PROGRAM PG_Regen
VAR
	Regenmacher: FB_Regenmacher;;
	Wetterbericht: FB_Wetterbericht;
END_VAR
VAR // added by the converter: edge detectors and wires of the graphical bodies
    _w1 : ANY;
END_VAR

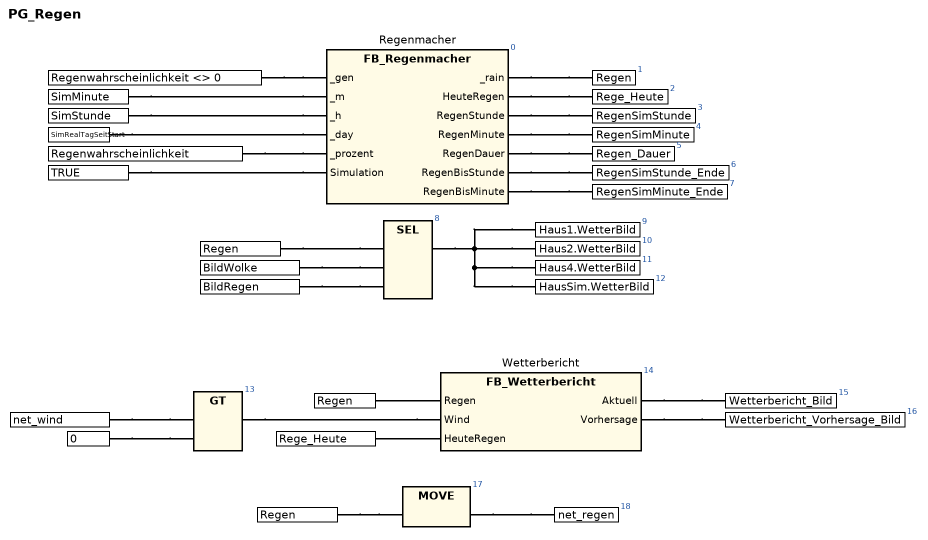
Regenmacher(
    _gen := Regenwahrscheinlichkeit <> 0,
    _m := SimMinute,
    _h := SimStunde,
    _day := SimRealTagSeitStart,
    _prozent := Regenwahrscheinlichkeit,
    Simulation := TRUE); // FB_Regenmacher
Regen := Regenmacher._rain;
Rege_Heute := Regenmacher.HeuteRegen;
RegenSimStunde := Regenmacher.RegenStunde;
RegenSimMinute := Regenmacher.RegenMinute;
Regen_Dauer := Regenmacher.RegenDauer;
RegenSimStunde_Ende := Regenmacher.RegenBisStunde;
RegenSimMinute_Ende := Regenmacher.RegenBisMinute;
_w1 := SEL(Regen, BildWolke, BildRegen);
Haus1.WetterBild := _w1;
Haus2.WetterBild := _w1;
Haus4.WetterBild := _w1;
HausSim.WetterBild := _w1;
Wetterbericht(Regen := Regen, Wind := net_wind > 0, HeuteRegen := Rege_Heute); // FB_Wetterbericht
Wetterbericht_Bild := Wetterbericht.Aktuell;
Wetterbericht_Vorhersage_Bild := Wetterbericht.Vorhersage;
net_regen := Regen;

END_PROGRAM

(* stored: Version 1.1.0.1, ProductVersion 3.1.4018.5
   POU PG_Regen: Id {adb02757-c25f-4f7e-abb3-6e14f23bc446}, SpecialFunc None *)
